(* Logix 5000 project; controller WP_Ottawa_Data_Concentrator_1 vendor 1 type 14 code 167 rev 32.14; software revision 32.04; part 2 of 5 *)
(* tags used below, declared in another part *)
   Break1_Length : DINT;
   Break2_Length : DINT;
   Lunch_Length : DINT;
   PreviousCount : DINT;
   Shift_Reset : BOOL;
   Shift_Reset_ONS : BOOL;
   LN31_Current_Shift_Duration_Mins : DINT;
   LN31_Current_Shift_Duration_wBreaks_Mins : DINT;
   LN31_DC_Controlled_Theoretical_Units : BOOL;
   LN31_Schedule : UDT_Current_Status;
   LN31_Schedule_Cycle_Timer : TIMER;
   LN31_Schedule_Max_Break_Duration : DINT;
   LN31_Schedule_Max_Break_Timer : TIMER;
   LN31_Schedule_TAKT : REAL;
   LN31_ScheduleUnits_Produced_from_line : DINT;
   LN31_Theoretical_Units_Counter : COUNTER;
   LN31_Theoretical_Units_Counter_ONS : BOOL;
   LN31_Weekly_Schedule : UDT_Weekly_Schedule;
   LN31_WorkstationsOA : DINT[120];
   null : STRING;
   Previous_Shift_Count : DINT;
(* LN31, continued *)

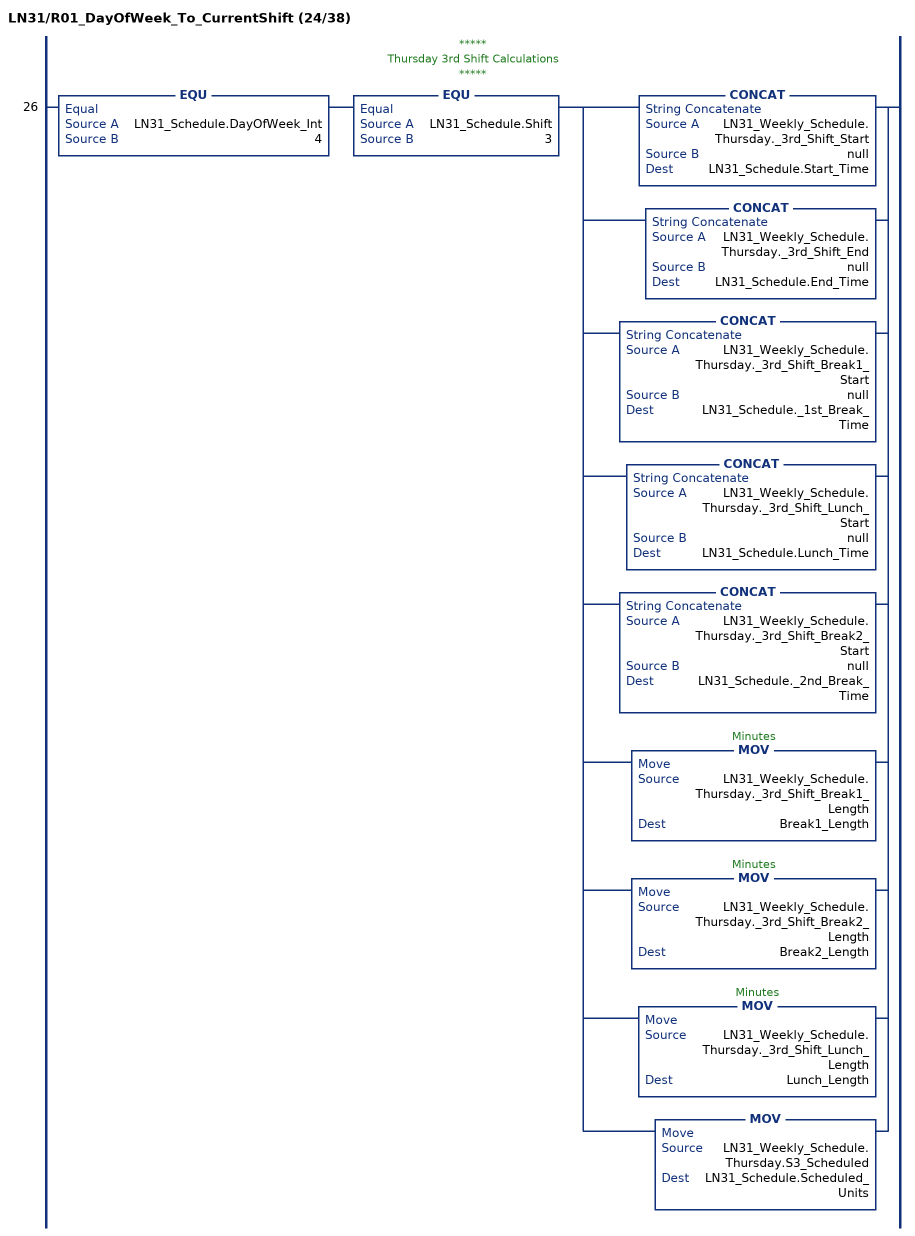
   [picture p24: LN31/R01_DayOfWeek_To_CurrentShift rungs 26-26]
   // *****
   // Thursday 3rd Shift Calculations
   // *****
   26: EQU(LN31_Schedule.DayOfWeek_Int,4)EQU(LN31_Schedule.Shift,3)[CONCAT(LN31_Weekly_Schedule.Thursday._3rd_Shift_Start,null,LN31_Schedule.Start_Time) ,CONCAT(LN31_Weekly_Schedule.Thursday._3rd_Shift_End,null,LN31_Schedule.End_Time) ,CONCAT(LN31_Weekly_Schedule.Thursday._3rd_Shift_Break1_Start,null,LN31_Schedule._1st_Break_Time) ,CONCAT(LN31_Weekly_Schedule.Thursday._3rd_Shift_Lunch_Start,null,LN31_Schedule.Lunch_Time) ,CONCAT(LN31_Weekly_Schedule.Thursday._3rd_Shift_Break2_Start,null,LN31_Schedule._2nd_Break_Time) ,MOV(LN31_Weekly_Schedule.Thursday._3rd_Shift_Break1_Length,Break1_Length) ,MOV(LN31_Weekly_Schedule.Thursday._3rd_Shift_Break2_Length,Break2_Length) ,MOV(LN31_Weekly_Schedule.Thursday._3rd_Shift_Lunch_Length,Lunch_Length) ,MOV(LN31_Weekly_Schedule.Thursday.S3_Scheduled,LN31_Schedule.Scheduled_Units) ];
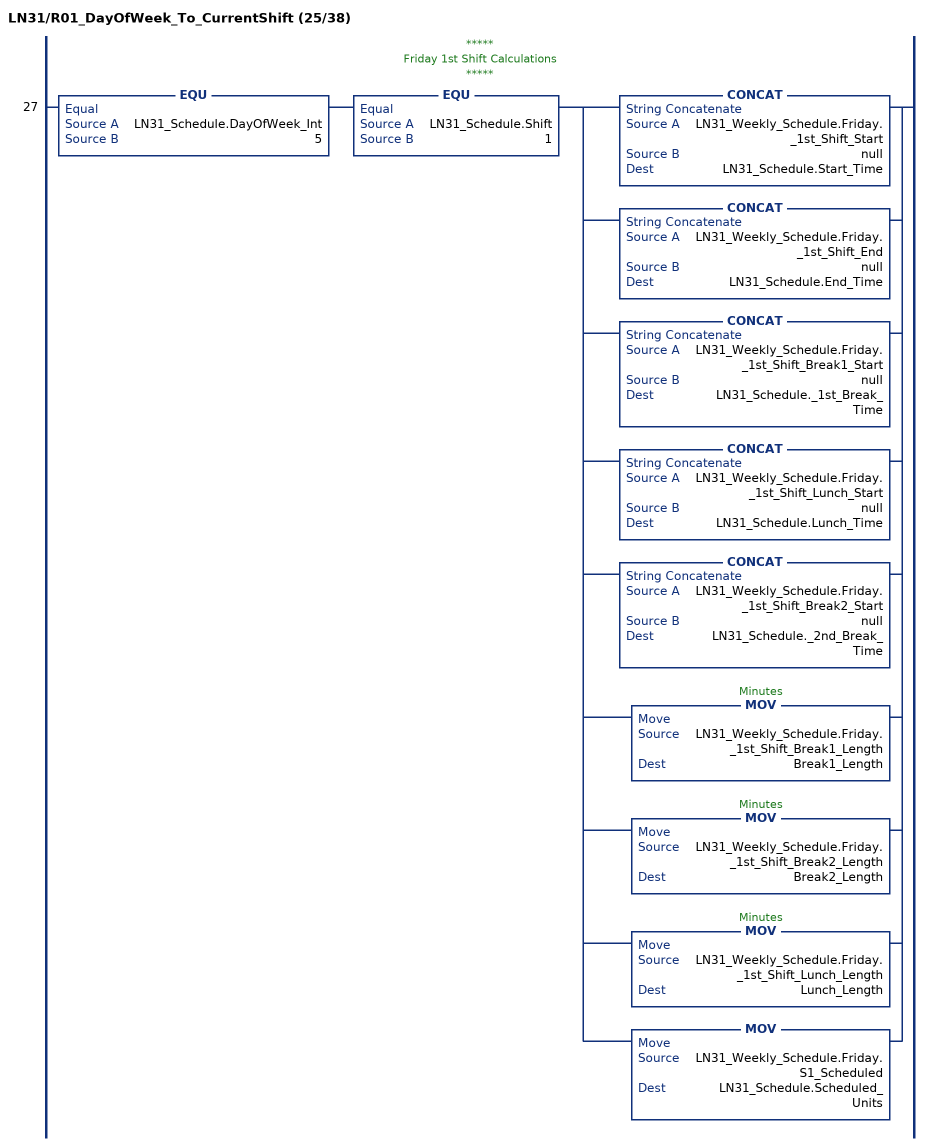
   // *****
   // Friday 1st Shift Calculations
   // *****
   27: EQU(LN31_Schedule.DayOfWeek_Int,5)EQU(LN31_Schedule.Shift,1)[CONCAT(LN31_Weekly_Schedule.Friday._1st_Shift_Start,null,LN31_Schedule.Start_Time) ,CONCAT(LN31_Weekly_Schedule.Friday._1st_Shift_End,null,LN31_Schedule.End_Time) ,CONCAT(LN31_Weekly_Schedule.Friday._1st_Shift_Break1_Start,null,LN31_Schedule._1st_Break_Time) ,CONCAT(LN31_Weekly_Schedule.Friday._1st_Shift_Lunch_Start,null,LN31_Schedule.Lunch_Time) ,CONCAT(LN31_Weekly_Schedule.Friday._1st_Shift_Break2_Start,null,LN31_Schedule._2nd_Break_Time) ,MOV(LN31_Weekly_Schedule.Friday._1st_Shift_Break1_Length,Break1_Length) ,MOV(LN31_Weekly_Schedule.Friday._1st_Shift_Break2_Length,Break2_Length) ,MOV(LN31_Weekly_Schedule.Friday._1st_Shift_Lunch_Length,Lunch_Length) ,MOV(LN31_Weekly_Schedule.Friday.S1_Scheduled,LN31_Schedule.Scheduled_Units) ];
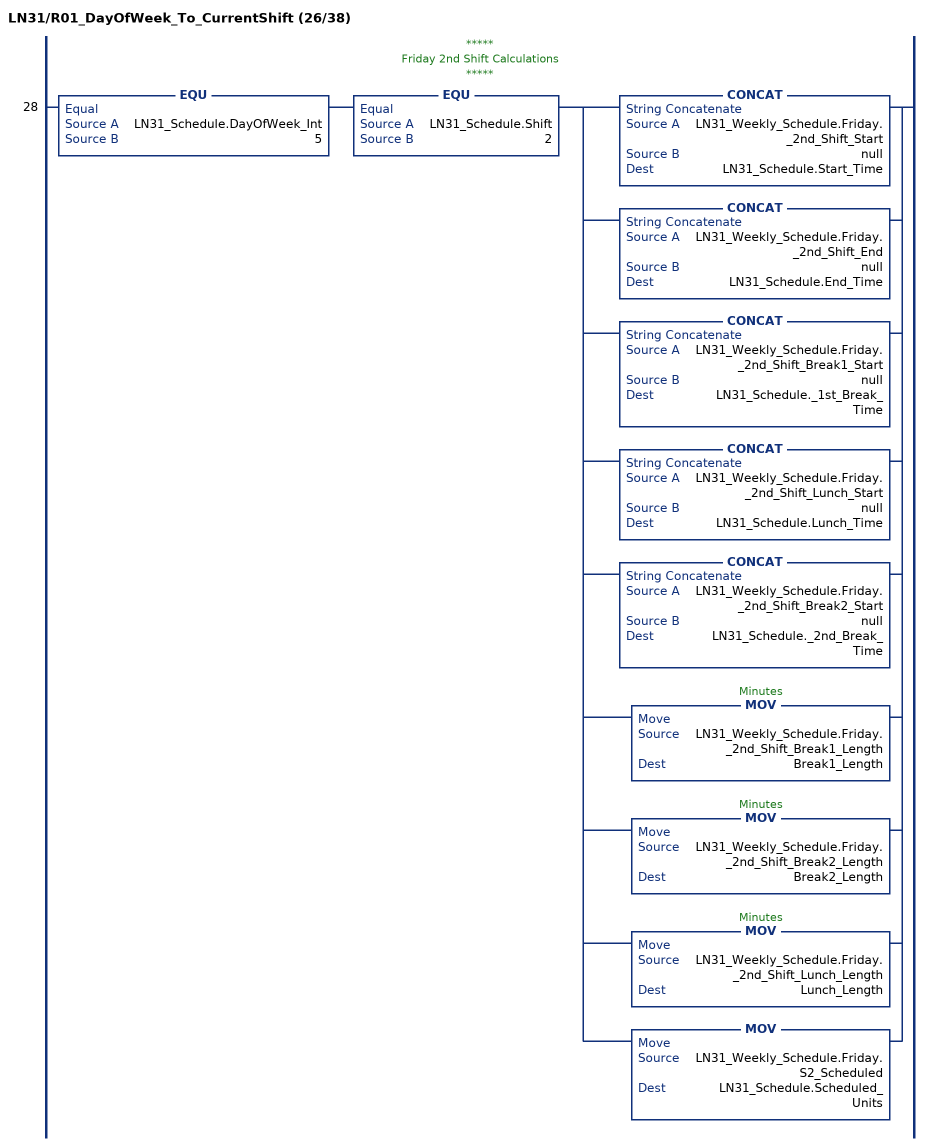
   // *****
   // Friday 2nd Shift Calculations
   // *****
   28: EQU(LN31_Schedule.DayOfWeek_Int,5)EQU(LN31_Schedule.Shift,2)[CONCAT(LN31_Weekly_Schedule.Friday._2nd_Shift_Start,null,LN31_Schedule.Start_Time) ,CONCAT(LN31_Weekly_Schedule.Friday._2nd_Shift_End,null,LN31_Schedule.End_Time) ,CONCAT(LN31_Weekly_Schedule.Friday._2nd_Shift_Break1_Start,null,LN31_Schedule._1st_Break_Time) ,CONCAT(LN31_Weekly_Schedule.Friday._2nd_Shift_Lunch_Start,null,LN31_Schedule.Lunch_Time) ,CONCAT(LN31_Weekly_Schedule.Friday._2nd_Shift_Break2_Start,null,LN31_Schedule._2nd_Break_Time) ,MOV(LN31_Weekly_Schedule.Friday._2nd_Shift_Break1_Length,Break1_Length) ,MOV(LN31_Weekly_Schedule.Friday._2nd_Shift_Break2_Length,Break2_Length) ,MOV(LN31_Weekly_Schedule.Friday._2nd_Shift_Lunch_Length,Lunch_Length) ,MOV(LN31_Weekly_Schedule.Friday.S2_Scheduled,LN31_Schedule.Scheduled_Units) ];
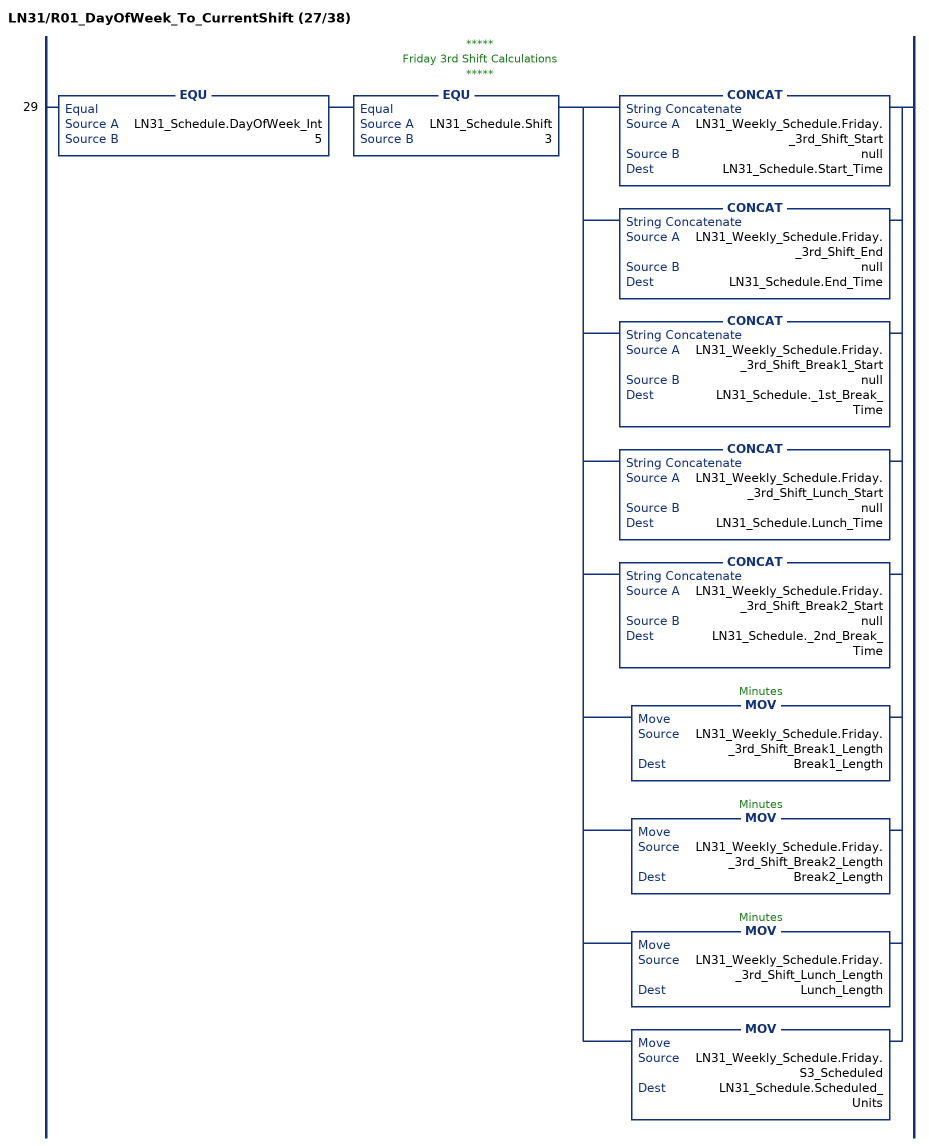
   // *****
   // Friday 3rd Shift Calculations
   // *****
   29: EQU(LN31_Schedule.DayOfWeek_Int,5)EQU(LN31_Schedule.Shift,3)[CONCAT(LN31_Weekly_Schedule.Friday._3rd_Shift_Start,null,LN31_Schedule.Start_Time) ,CONCAT(LN31_Weekly_Schedule.Friday._3rd_Shift_End,null,LN31_Schedule.End_Time) ,CONCAT(LN31_Weekly_Schedule.Friday._3rd_Shift_Break1_Start,null,LN31_Schedule._1st_Break_Time) ,CONCAT(LN31_Weekly_Schedule.Friday._3rd_Shift_Lunch_Start,null,LN31_Schedule.Lunch_Time) ,CONCAT(LN31_Weekly_Schedule.Friday._3rd_Shift_Break2_Start,null,LN31_Schedule._2nd_Break_Time) ,MOV(LN31_Weekly_Schedule.Friday._3rd_Shift_Break1_Length,Break1_Length) ,MOV(LN31_Weekly_Schedule.Friday._3rd_Shift_Break2_Length,Break2_Length) ,MOV(LN31_Weekly_Schedule.Friday._3rd_Shift_Lunch_Length,Lunch_Length) ,MOV(LN31_Weekly_Schedule.Friday.S3_Scheduled,LN31_Schedule.Scheduled_Units) ];
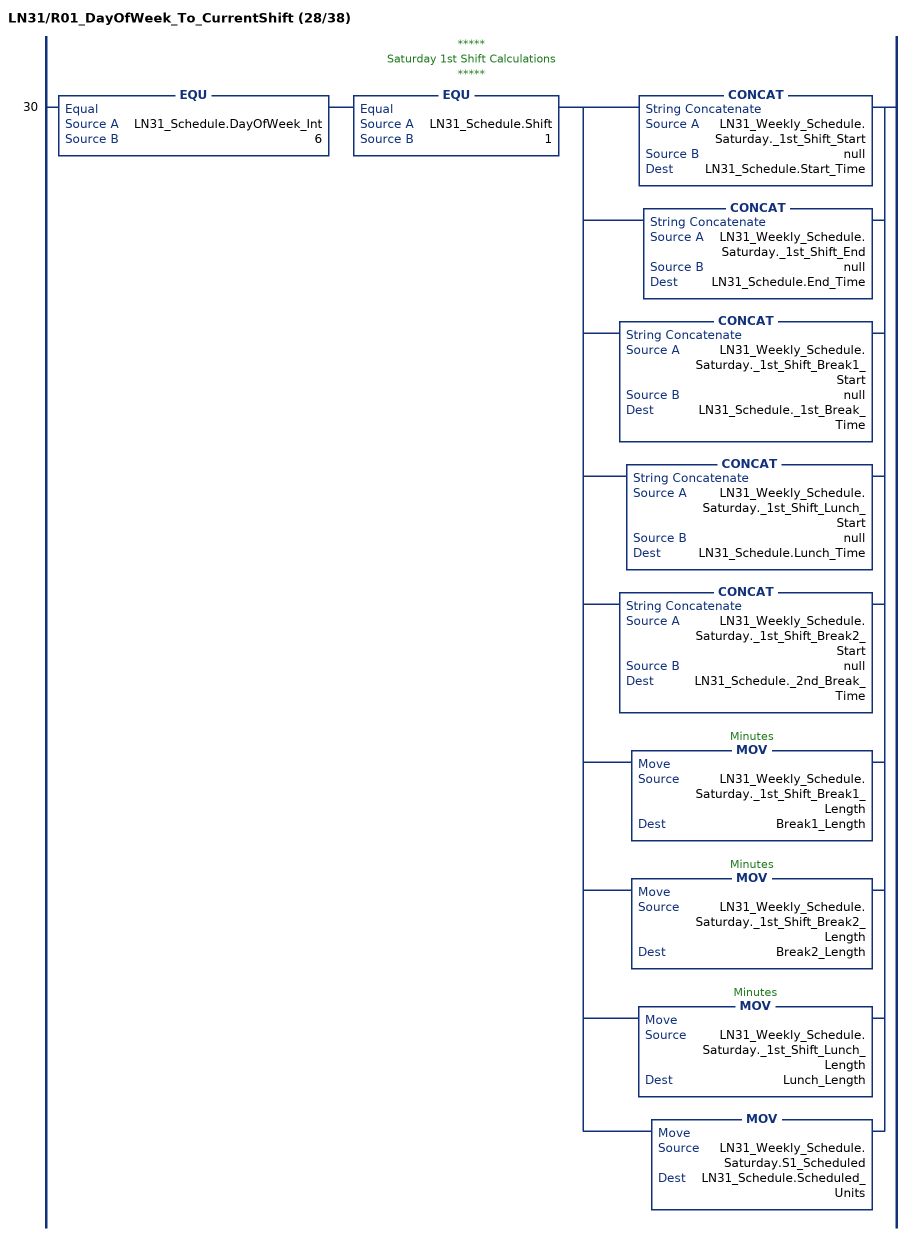
   // *****
   // Saturday 1st Shift Calculations
   // *****
   30: EQU(LN31_Schedule.DayOfWeek_Int,6)EQU(LN31_Schedule.Shift,1)[CONCAT(LN31_Weekly_Schedule.Saturday._1st_Shift_Start,null,LN31_Schedule.Start_Time) ,CONCAT(LN31_Weekly_Schedule.Saturday._1st_Shift_End,null,LN31_Schedule.End_Time) ,CONCAT(LN31_Weekly_Schedule.Saturday._1st_Shift_Break1_Start,null,LN31_Schedule._1st_Break_Time) ,CONCAT(LN31_Weekly_Schedule.Saturday._1st_Shift_Lunch_Start,null,LN31_Schedule.Lunch_Time) ,CONCAT(LN31_Weekly_Schedule.Saturday._1st_Shift_Break2_Start,null,LN31_Schedule._2nd_Break_Time) ,MOV(LN31_Weekly_Schedule.Saturday._1st_Shift_Break1_Length,Break1_Length) ,MOV(LN31_Weekly_Schedule.Saturday._1st_Shift_Break2_Length,Break2_Length) ,MOV(LN31_Weekly_Schedule.Saturday._1st_Shift_Lunch_Length,Lunch_Length) ,MOV(LN31_Weekly_Schedule.Saturday.S1_Scheduled,LN31_Schedule.Scheduled_Units) ];
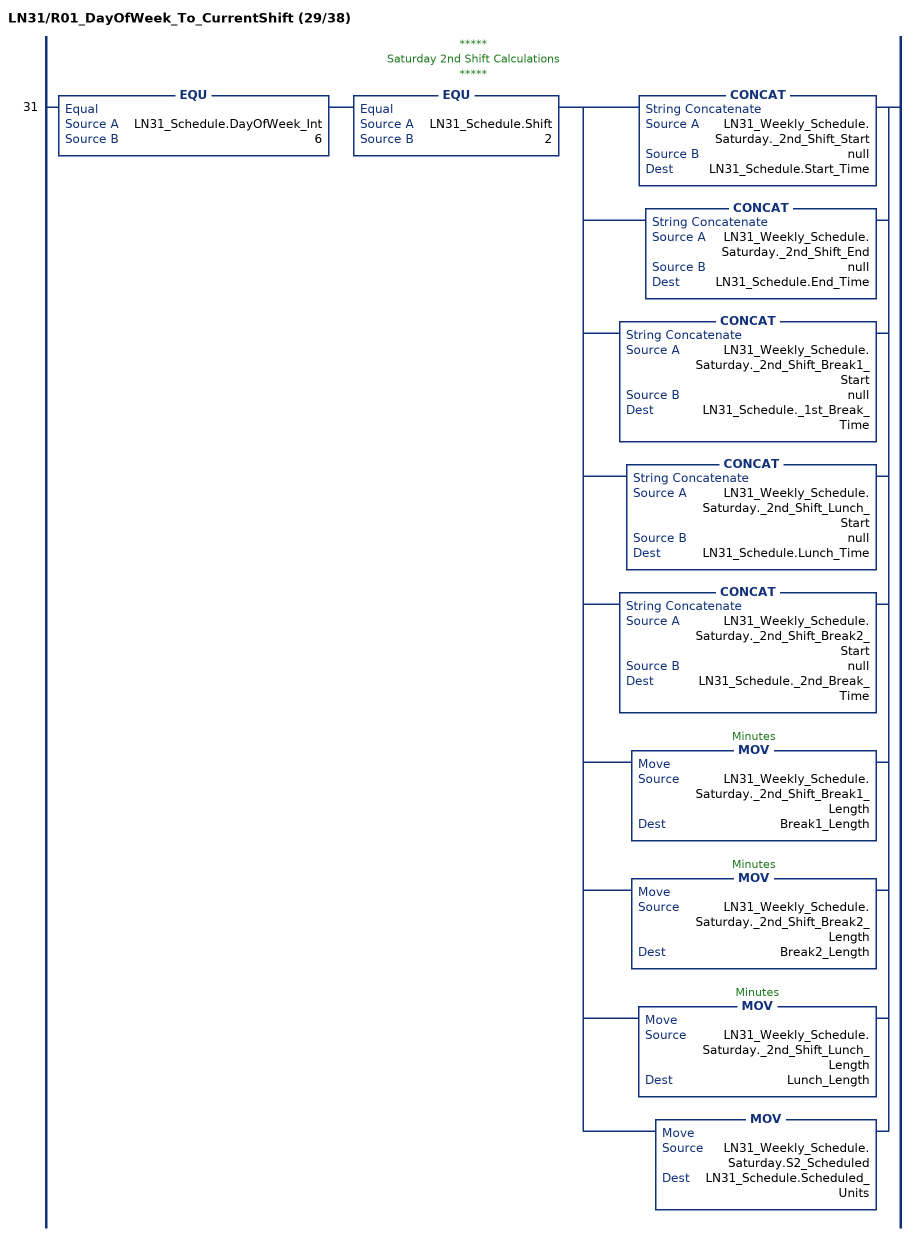
   // *****
   // Saturday 2nd Shift Calculations
   // *****
   31: EQU(LN31_Schedule.DayOfWeek_Int,6)EQU(LN31_Schedule.Shift,2)[CONCAT(LN31_Weekly_Schedule.Saturday._2nd_Shift_Start,null,LN31_Schedule.Start_Time) ,CONCAT(LN31_Weekly_Schedule.Saturday._2nd_Shift_End,null,LN31_Schedule.End_Time) ,CONCAT(LN31_Weekly_Schedule.Saturday._2nd_Shift_Break1_Start,null,LN31_Schedule._1st_Break_Time) ,CONCAT(LN31_Weekly_Schedule.Saturday._2nd_Shift_Lunch_Start,null,LN31_Schedule.Lunch_Time) ,CONCAT(LN31_Weekly_Schedule.Saturday._2nd_Shift_Break2_Start,null,LN31_Schedule._2nd_Break_Time) ,MOV(LN31_Weekly_Schedule.Saturday._2nd_Shift_Break1_Length,Break1_Length) ,MOV(LN31_Weekly_Schedule.Saturday._2nd_Shift_Break2_Length,Break2_Length) ,MOV(LN31_Weekly_Schedule.Saturday._2nd_Shift_Lunch_Length,Lunch_Length) ,MOV(LN31_Weekly_Schedule.Saturday.S2_Scheduled,LN31_Schedule.Scheduled_Units) ];
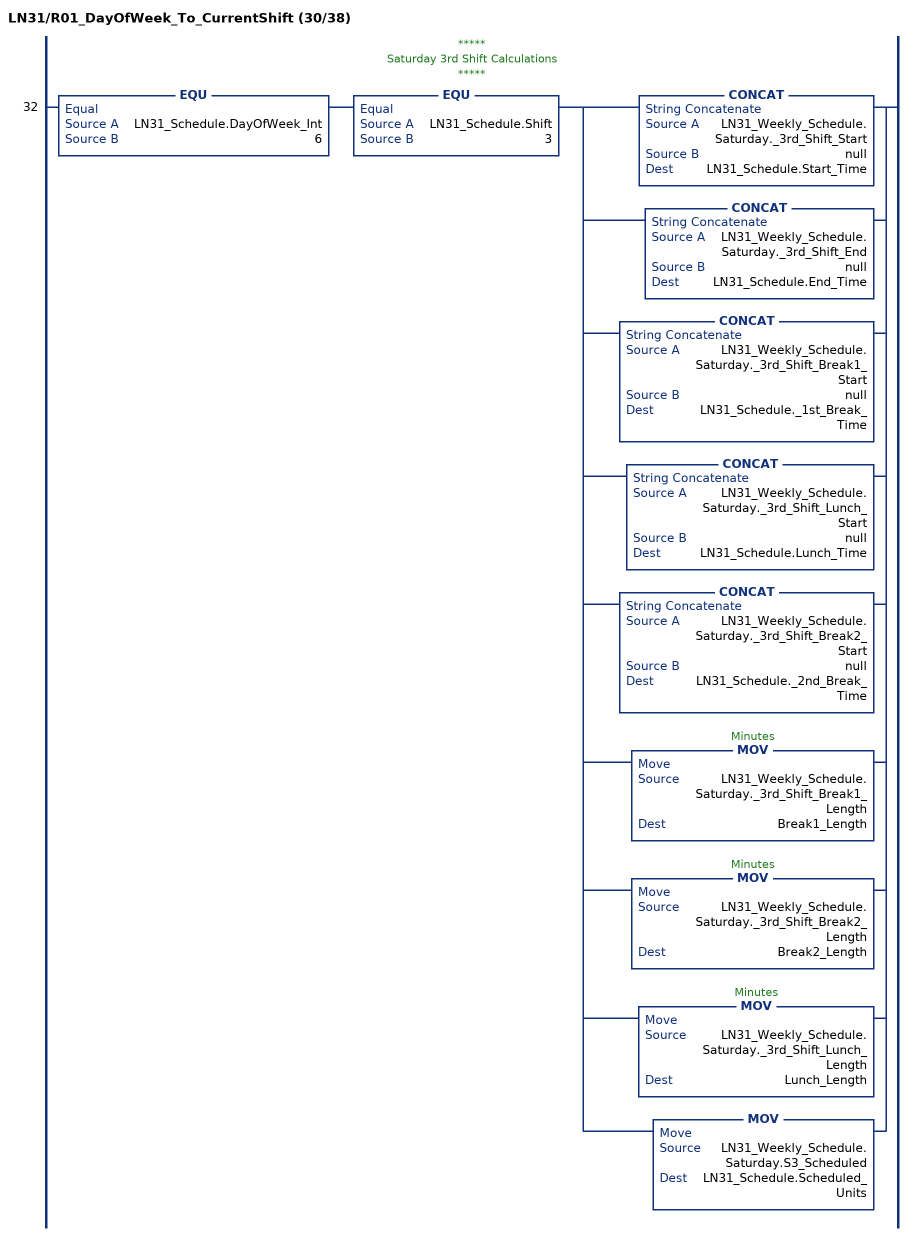
   // *****
   // Saturday 3rd Shift Calculations
   // *****
   32: EQU(LN31_Schedule.DayOfWeek_Int,6)EQU(LN31_Schedule.Shift,3)[CONCAT(LN31_Weekly_Schedule.Saturday._3rd_Shift_Start,null,LN31_Schedule.Start_Time) ,CONCAT(LN31_Weekly_Schedule.Saturday._3rd_Shift_End,null,LN31_Schedule.End_Time) ,CONCAT(LN31_Weekly_Schedule.Saturday._3rd_Shift_Break1_Start,null,LN31_Schedule._1st_Break_Time) ,CONCAT(LN31_Weekly_Schedule.Saturday._3rd_Shift_Lunch_Start,null,LN31_Schedule.Lunch_Time) ,CONCAT(LN31_Weekly_Schedule.Saturday._3rd_Shift_Break2_Start,null,LN31_Schedule._2nd_Break_Time) ,MOV(LN31_Weekly_Schedule.Saturday._3rd_Shift_Break1_Length,Break1_Length) ,MOV(LN31_Weekly_Schedule.Saturday._3rd_Shift_Break2_Length,Break2_Length) ,MOV(LN31_Weekly_Schedule.Saturday._3rd_Shift_Lunch_Length,Lunch_Length) ,MOV(LN31_Weekly_Schedule.Saturday.S3_Scheduled,LN31_Schedule.Scheduled_Units) ];
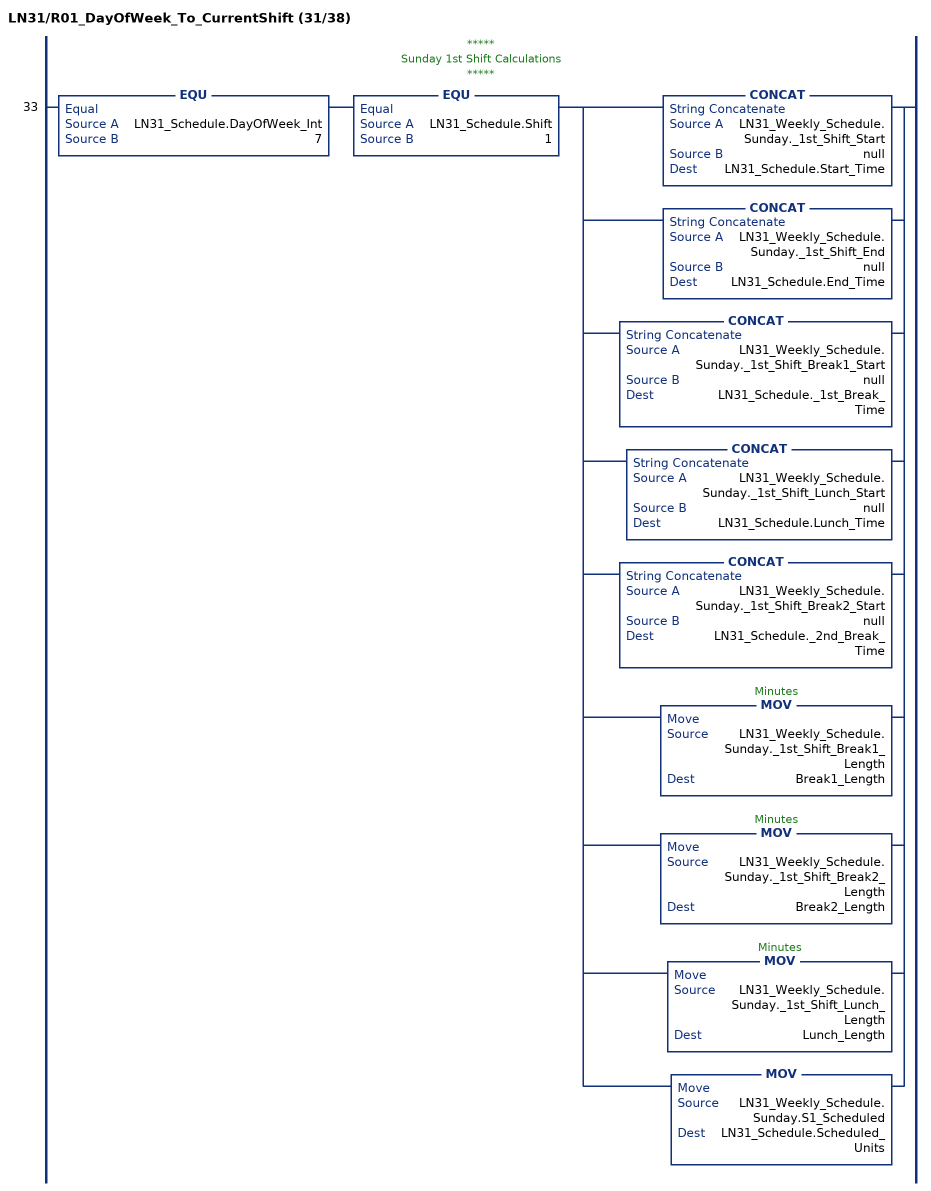
   // *****
   // Sunday 1st Shift Calculations
   // *****
   33: EQU(LN31_Schedule.DayOfWeek_Int,7)EQU(LN31_Schedule.Shift,1)[CONCAT(LN31_Weekly_Schedule.Sunday._1st_Shift_Start,null,LN31_Schedule.Start_Time) ,CONCAT(LN31_Weekly_Schedule.Sunday._1st_Shift_End,null,LN31_Schedule.End_Time) ,CONCAT(LN31_Weekly_Schedule.Sunday._1st_Shift_Break1_Start,null,LN31_Schedule._1st_Break_Time) ,CONCAT(LN31_Weekly_Schedule.Sunday._1st_Shift_Lunch_Start,null,LN31_Schedule.Lunch_Time) ,CONCAT(LN31_Weekly_Schedule.Sunday._1st_Shift_Break2_Start,null,LN31_Schedule._2nd_Break_Time) ,MOV(LN31_Weekly_Schedule.Sunday._1st_Shift_Break1_Length,Break1_Length) ,MOV(LN31_Weekly_Schedule.Sunday._1st_Shift_Break2_Length,Break2_Length) ,MOV(LN31_Weekly_Schedule.Sunday._1st_Shift_Lunch_Length,Lunch_Length) ,MOV(LN31_Weekly_Schedule.Sunday.S1_Scheduled,LN31_Schedule.Scheduled_Units) ];
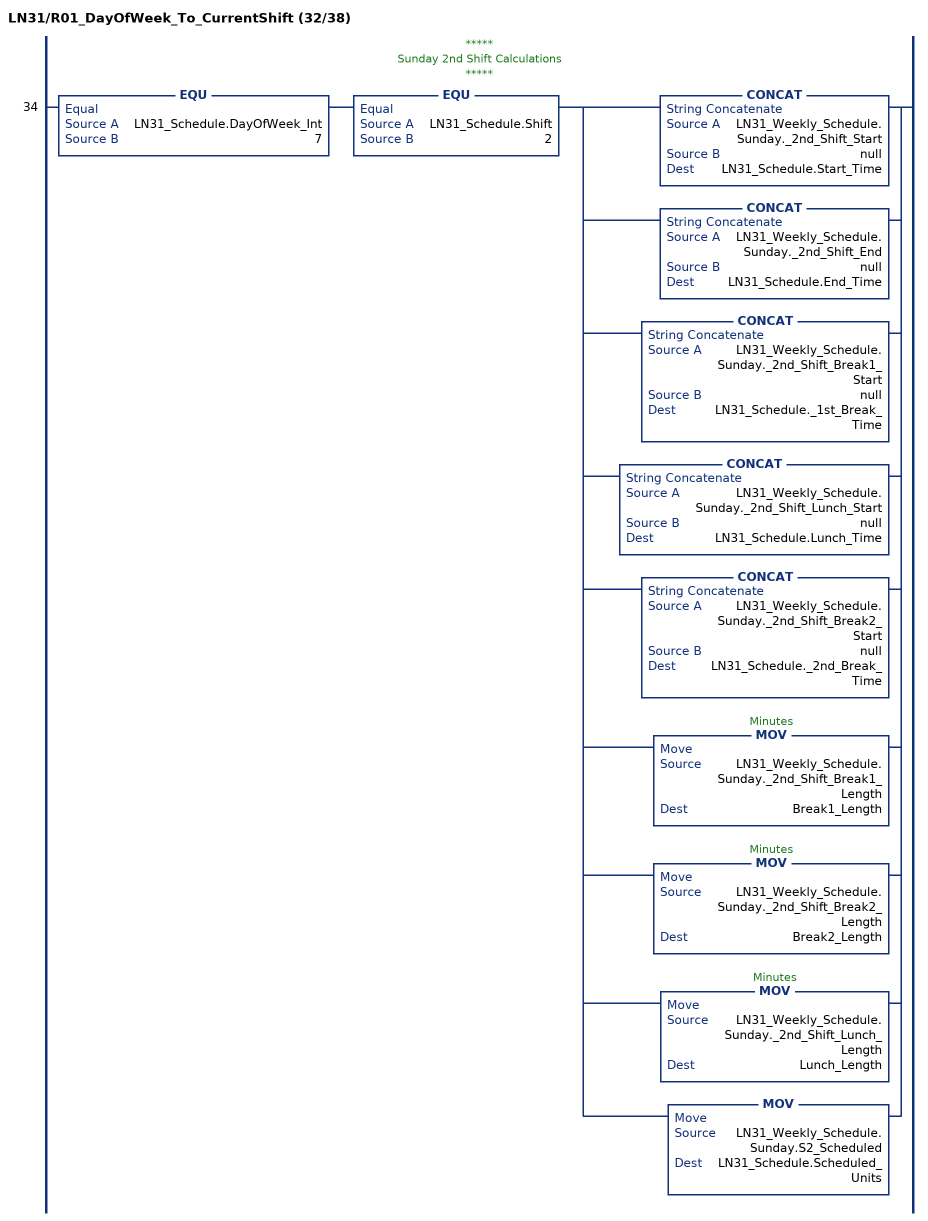
   // *****
   // Sunday 2nd Shift Calculations
   // *****
   34: EQU(LN31_Schedule.DayOfWeek_Int,7)EQU(LN31_Schedule.Shift,2)[CONCAT(LN31_Weekly_Schedule.Sunday._2nd_Shift_Start,null,LN31_Schedule.Start_Time) ,CONCAT(LN31_Weekly_Schedule.Sunday._2nd_Shift_End,null,LN31_Schedule.End_Time) ,CONCAT(LN31_Weekly_Schedule.Sunday._2nd_Shift_Break1_Start,null,LN31_Schedule._1st_Break_Time) ,CONCAT(LN31_Weekly_Schedule.Sunday._2nd_Shift_Lunch_Start,null,LN31_Schedule.Lunch_Time) ,CONCAT(LN31_Weekly_Schedule.Sunday._2nd_Shift_Break2_Start,null,LN31_Schedule._2nd_Break_Time) ,MOV(LN31_Weekly_Schedule.Sunday._2nd_Shift_Break1_Length,Break1_Length) ,MOV(LN31_Weekly_Schedule.Sunday._2nd_Shift_Break2_Length,Break2_Length) ,MOV(LN31_Weekly_Schedule.Sunday._2nd_Shift_Lunch_Length,Lunch_Length) ,MOV(LN31_Weekly_Schedule.Sunday.S2_Scheduled,LN31_Schedule.Scheduled_Units) ];
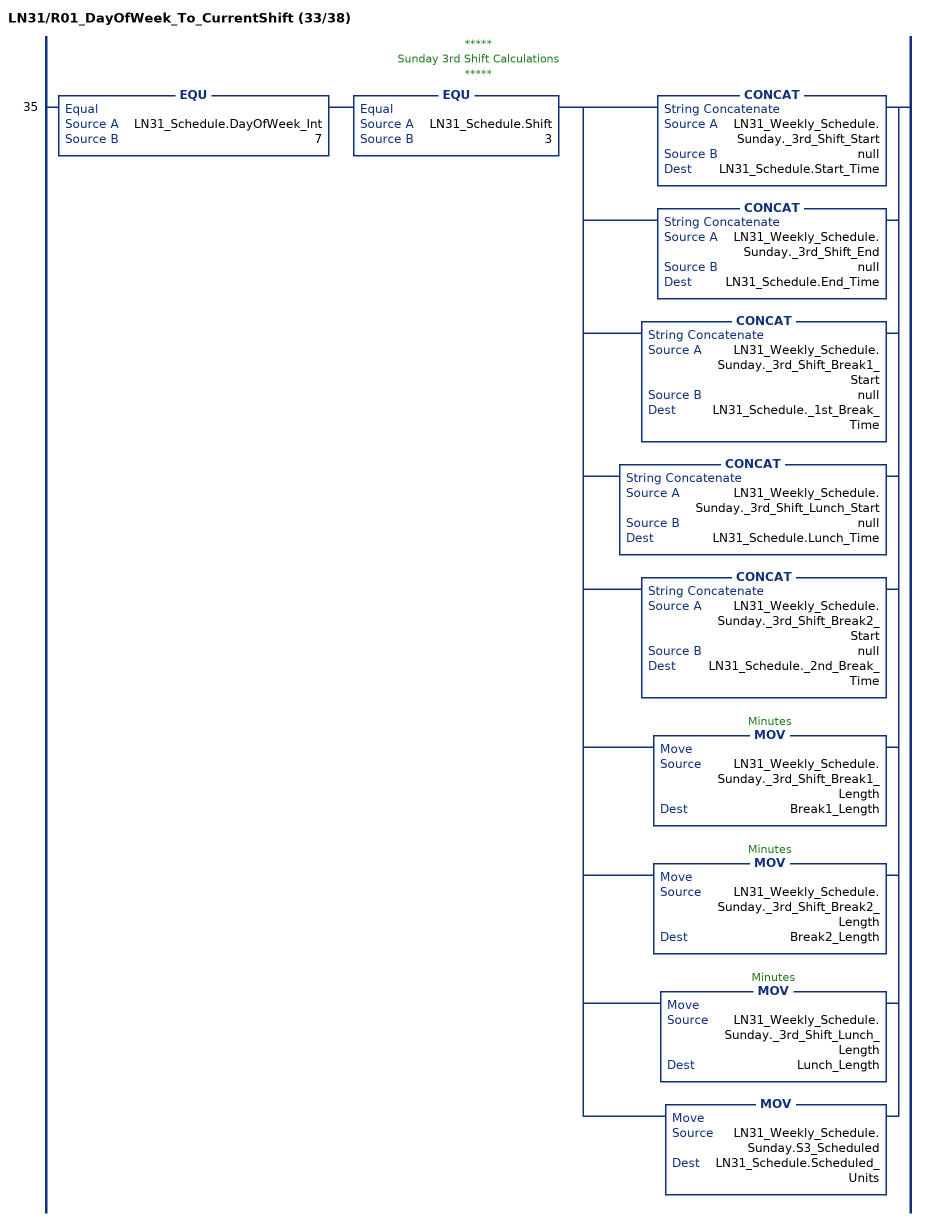
   // *****
   // Sunday 3rd Shift Calculations
   // *****
   35: EQU(LN31_Schedule.DayOfWeek_Int,7)EQU(LN31_Schedule.Shift,3)[CONCAT(LN31_Weekly_Schedule.Sunday._3rd_Shift_Start,null,LN31_Schedule.Start_Time) ,CONCAT(LN31_Weekly_Schedule.Sunday._3rd_Shift_End,null,LN31_Schedule.End_Time) ,CONCAT(LN31_Weekly_Schedule.Sunday._3rd_Shift_Break1_Start,null,LN31_Schedule._1st_Break_Time) ,CONCAT(LN31_Weekly_Schedule.Sunday._3rd_Shift_Lunch_Start,null,LN31_Schedule.Lunch_Time) ,CONCAT(LN31_Weekly_Schedule.Sunday._3rd_Shift_Break2_Start,null,LN31_Schedule._2nd_Break_Time) ,MOV(LN31_Weekly_Schedule.Sunday._3rd_Shift_Break1_Length,Break1_Length) ,MOV(LN31_Weekly_Schedule.Sunday._3rd_Shift_Break2_Length,Break2_Length) ,MOV(LN31_Weekly_Schedule.Sunday._3rd_Shift_Lunch_Length,Lunch_Length) ,MOV(LN31_Weekly_Schedule.Sunday.S3_Scheduled,LN31_Schedule.Scheduled_Units) ];
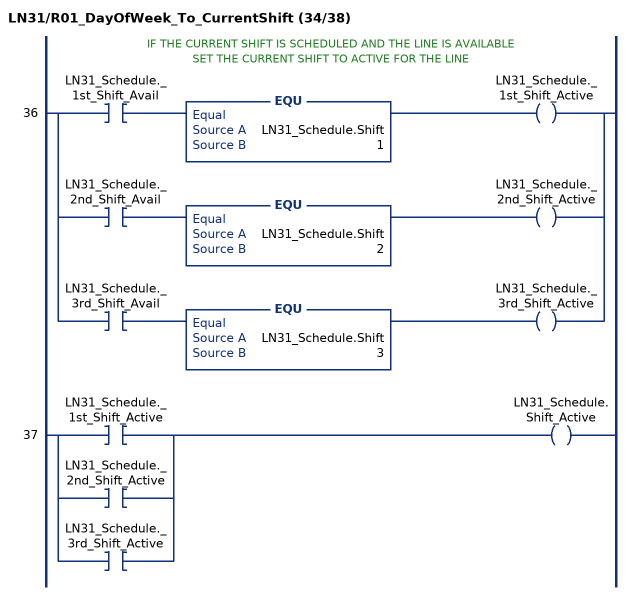
   // IF THE CURRENT SHIFT IS SCHEDULED AND THE LINE IS AVAILABLE
   // SET THE CURRENT SHIFT TO ACTIVE FOR THE LINE
   36: [XIC(LN31_Schedule._1st_Shift_Avail) EQU(LN31_Schedule.Shift,1) OTE(LN31_Schedule._1st_Shift_Active) ,XIC(LN31_Schedule._2nd_Shift_Avail) EQU(LN31_Schedule.Shift,2) OTE(LN31_Schedule._2nd_Shift_Active) ,XIC(LN31_Schedule._3rd_Shift_Avail) EQU(LN31_Schedule.Shift,3) OTE(LN31_Schedule._3rd_Shift_Active) ];
   37: [XIC(LN31_Schedule._1st_Shift_Active) ,XIC(LN31_Schedule._2nd_Shift_Active) ,XIC(LN31_Schedule._3rd_Shift_Active) ]OTE(LN31_Schedule.Shift_Active);
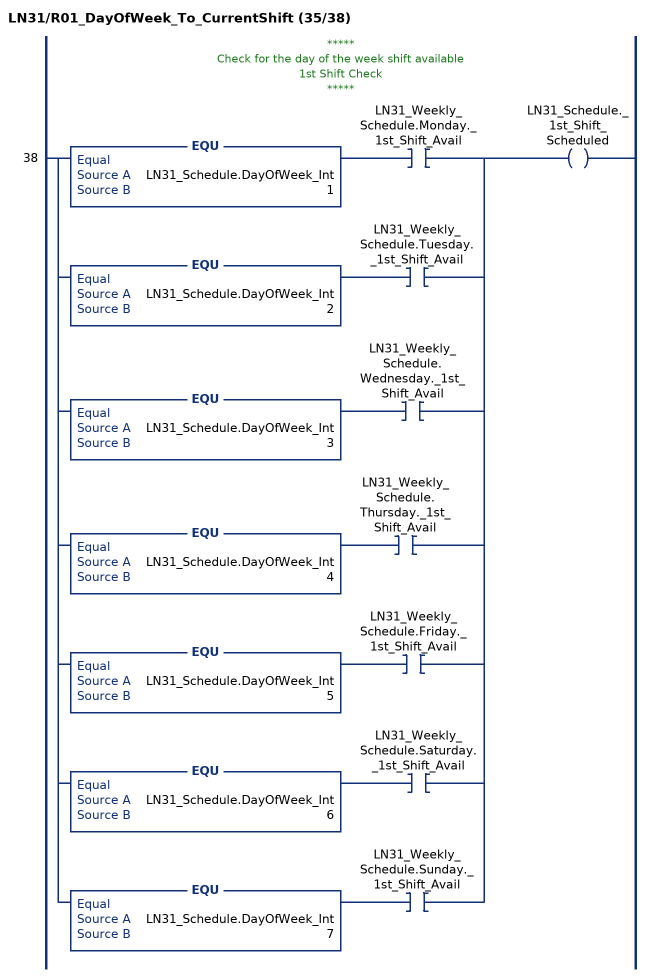
   // *****
   // Check for the day of the week shift available
   // 1st Shift Check
   // *****
   38: [EQU(LN31_Schedule.DayOfWeek_Int,1) XIC(LN31_Weekly_Schedule.Monday._1st_Shift_Avail) ,EQU(LN31_Schedule.DayOfWeek_Int,2) XIC(LN31_Weekly_Schedule.Tuesday._1st_Shift_Avail) ,EQU(LN31_Schedule.DayOfWeek_Int,3) XIC(LN31_Weekly_Schedule.Wednesday._1st_Shift_Avail) ,EQU(LN31_Schedule.DayOfWeek_Int,4) XIC(LN31_Weekly_Schedule.Thursday._1st_Shift_Avail) ,EQU(LN31_Schedule.DayOfWeek_Int,5) XIC(LN31_Weekly_Schedule.Friday._1st_Shift_Avail) ,EQU(LN31_Schedule.DayOfWeek_Int,6) XIC(LN31_Weekly_Schedule.Saturday._1st_Shift_Avail) ,EQU(LN31_Schedule.DayOfWeek_Int,7) XIC(LN31_Weekly_Schedule.Sunday._1st_Shift_Avail) ]OTE(LN31_Schedule._1st_Shift_Scheduled);
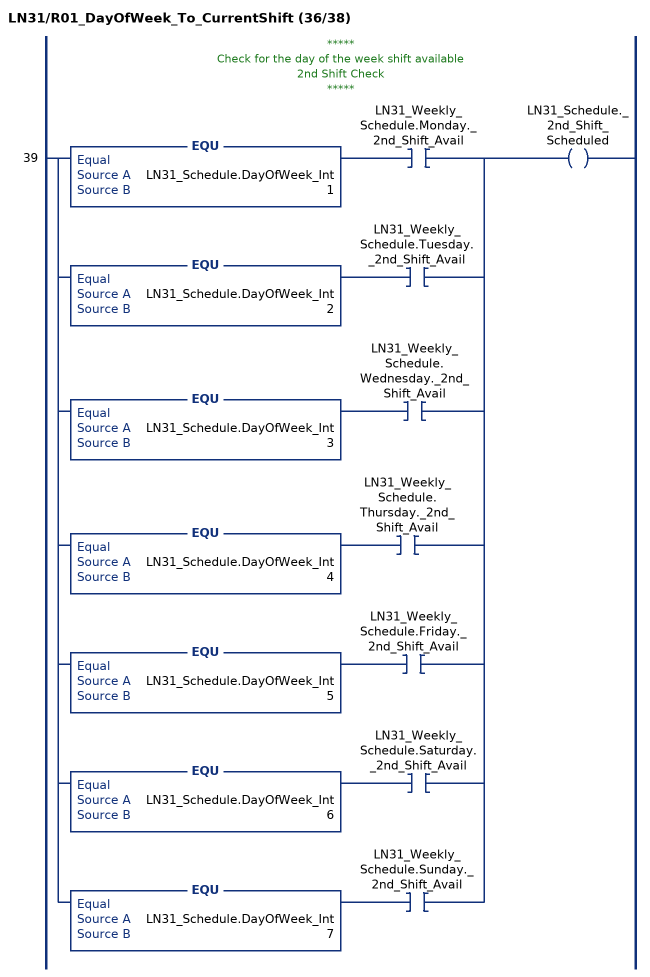
   // *****
   // Check for the day of the week shift available
   // 2nd Shift Check
   // *****
   39: [EQU(LN31_Schedule.DayOfWeek_Int,1) XIC(LN31_Weekly_Schedule.Monday._2nd_Shift_Avail) ,EQU(LN31_Schedule.DayOfWeek_Int,2) XIC(LN31_Weekly_Schedule.Tuesday._2nd_Shift_Avail) ,EQU(LN31_Schedule.DayOfWeek_Int,3) XIC(LN31_Weekly_Schedule.Wednesday._2nd_Shift_Avail) ,EQU(LN31_Schedule.DayOfWeek_Int,4) XIC(LN31_Weekly_Schedule.Thursday._2nd_Shift_Avail) ,EQU(LN31_Schedule.DayOfWeek_Int,5) XIC(LN31_Weekly_Schedule.Friday._2nd_Shift_Avail) ,EQU(LN31_Schedule.DayOfWeek_Int,6) XIC(LN31_Weekly_Schedule.Saturday._2nd_Shift_Avail) ,EQU(LN31_Schedule.DayOfWeek_Int,7) XIC(LN31_Weekly_Schedule.Sunday._2nd_Shift_Avail) ]OTE(LN31_Schedule._2nd_Shift_Scheduled);
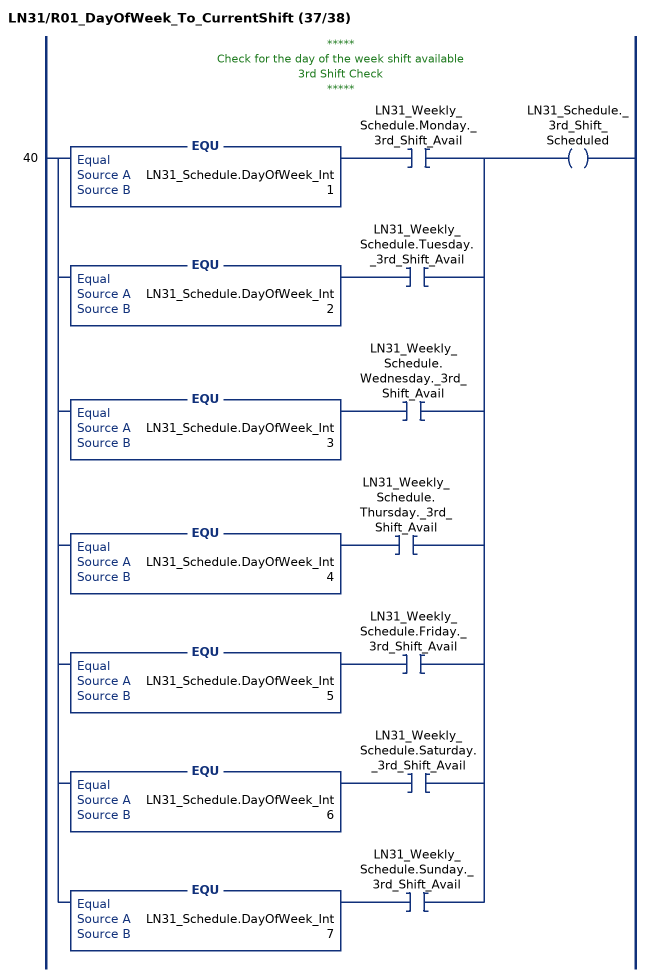
   // *****
   // Check for the day of the week shift available
   // 3rd Shift Check
   // *****
   40: [EQU(LN31_Schedule.DayOfWeek_Int,1) XIC(LN31_Weekly_Schedule.Monday._3rd_Shift_Avail) ,EQU(LN31_Schedule.DayOfWeek_Int,2) XIC(LN31_Weekly_Schedule.Tuesday._3rd_Shift_Avail) ,EQU(LN31_Schedule.DayOfWeek_Int,3) XIC(LN31_Weekly_Schedule.Wednesday._3rd_Shift_Avail) ,EQU(LN31_Schedule.DayOfWeek_Int,4) XIC(LN31_Weekly_Schedule.Thursday._3rd_Shift_Avail) ,EQU(LN31_Schedule.DayOfWeek_Int,5) XIC(LN31_Weekly_Schedule.Friday._3rd_Shift_Avail) ,EQU(LN31_Schedule.DayOfWeek_Int,6) XIC(LN31_Weekly_Schedule.Saturday._3rd_Shift_Avail) ,EQU(LN31_Schedule.DayOfWeek_Int,7) XIC(LN31_Weekly_Schedule.Sunday._3rd_Shift_Avail) ]OTE(LN31_Schedule._3rd_Shift_Scheduled);
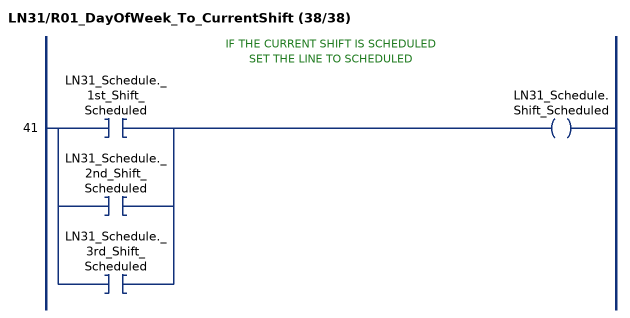
   // IF THE CURRENT SHIFT IS SCHEDULED
   // SET THE LINE TO SCHEDULED
   41: [XIC(LN31_Schedule._1st_Shift_Scheduled) ,XIC(LN31_Schedule._2nd_Shift_Scheduled) ,XIC(LN31_Schedule._3rd_Shift_Scheduled) ]OTE(LN31_Schedule.Shift_Scheduled);
END_ROUTINE

ROUTINE R02_CurrentShift_Calcs   (* ladder *)
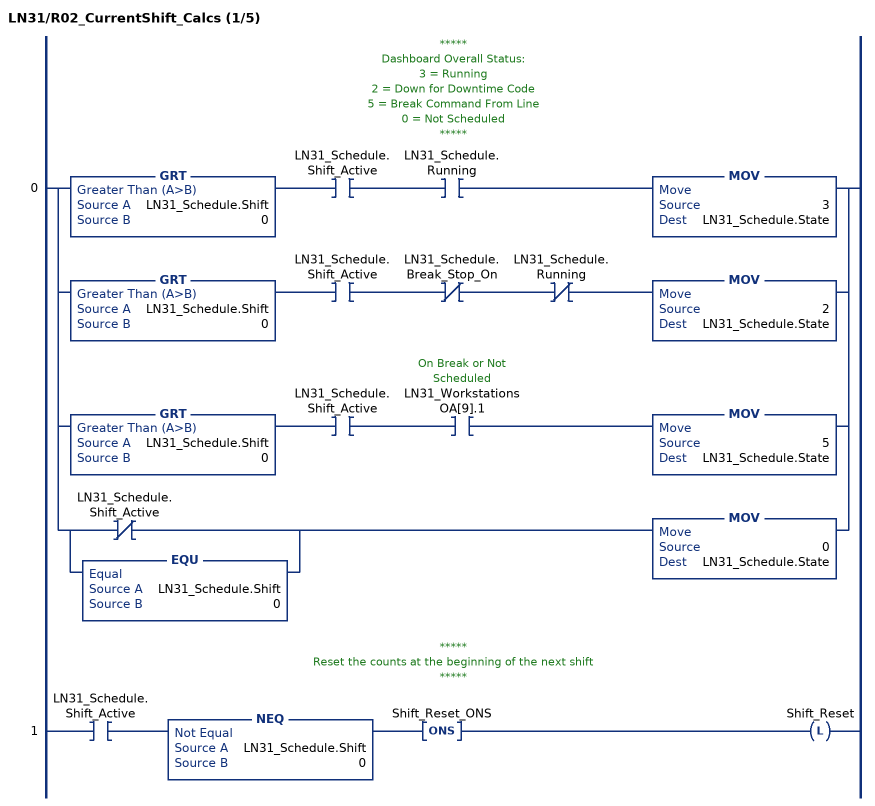
   // *****
   // Dashboard Overall Status:
   // 3 = Running
   // 2 = Down for Downtime Code
   // 5 = Break Command From Line
   // 0 = Not Scheduled
   // *****
   0: [GRT(LN31_Schedule.Shift,0) XIC(LN31_Schedule.Shift_Active) XIC(LN31_Schedule.Running) MOV(3,LN31_Schedule.State) ,GRT(LN31_Schedule.Shift,0) XIC(LN31_Schedule.Shift_Active) XIO(LN31_Schedule.Break_Stop_On) XIO(LN31_Schedule.Running) MOV(2,LN31_Schedule.State) ,GRT(LN31_Schedule.Shift,0) XIC(LN31_Schedule.Shift_Active) XIC(LN31_WorkstationsOA[9].1) MOV(5,LN31_Schedule.State) ,[XIO(LN31_Schedule.Shift_Active) ,EQU(LN31_Schedule.Shift,0) ] MOV(0,LN31_Schedule.State) ];
   // *****
   // Reset the counts at the beginning of the next shift
   // *****
   1: XIC(LN31_Schedule.Shift_Active)NEQ(LN31_Schedule.Shift,0)ONS(Shift_Reset_ONS)OTL(Shift_Reset);
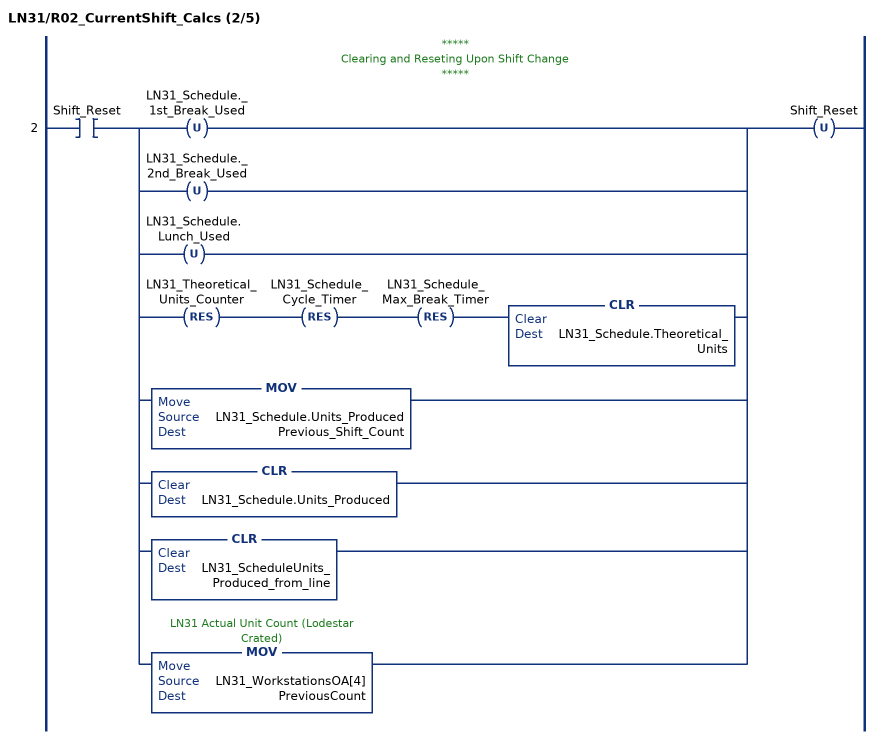
   // *****
   // Clearing and Reseting Upon Shift Change
   // *****
   2: XIC(Shift_Reset)[OTU(LN31_Schedule._1st_Break_Used) ,OTU(LN31_Schedule._2nd_Break_Used) ,OTU(LN31_Schedule.Lunch_Used) ,RES(LN31_Theoretical_Units_Counter) RES(LN31_Schedule_Cycle_Timer) RES(LN31_Schedule_Max_Break_Timer) CLR(LN31_Schedule.Theoretical_Units) ,MOV(LN31_Schedule.Units_Produced,Previous_Shift_Count) ,CLR(LN31_Schedule.Units_Produced) ,CLR(LN31_ScheduleUnits_Produced_from_line) ,MOV(LN31_WorkstationsOA[4],PreviousCount) ]OTU(Shift_Reset);
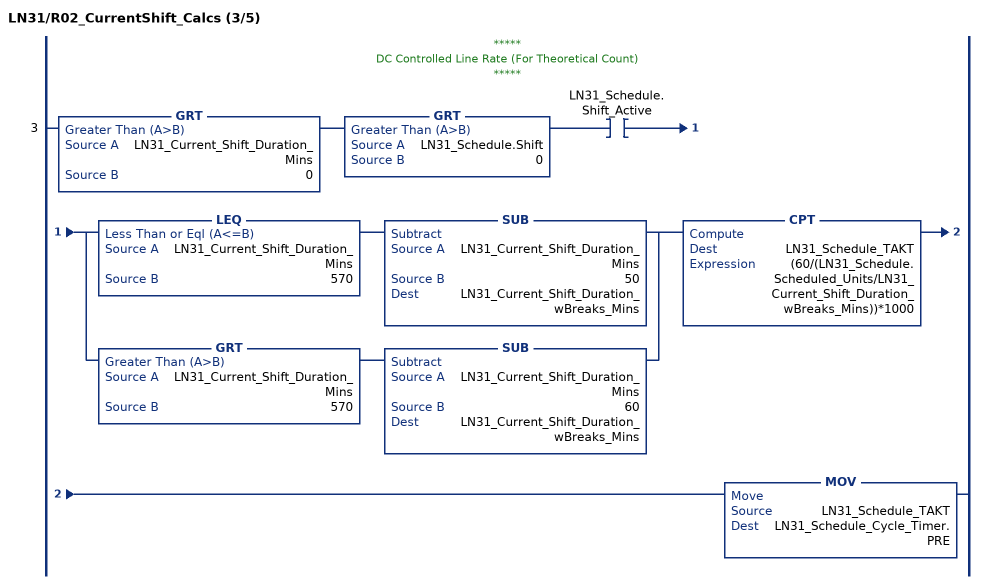
   // *****
   // DC Controlled Line Rate (For Theoretical Count)
   // *****
   3: GRT(LN31_Current_Shift_Duration_Mins,0)GRT(LN31_Schedule.Shift,0)XIC(LN31_Schedule.Shift_Active)[LEQ(LN31_Current_Shift_Duration_Mins,570) SUB(LN31_Current_Shift_Duration_Mins,50,LN31_Current_Shift_Duration_wBreaks_Mins) ,GRT(LN31_Current_Shift_Duration_Mins,570) SUB(LN31_Current_Shift_Duration_Mins,60,LN31_Current_Shift_Duration_wBreaks_Mins) ]CPT(LN31_Schedule_TAKT,(60/(LN31_Schedule.Scheduled_Units/LN31_Current_Shift_Duration_wBreaks_Mins))*1000)MOV(LN31_Schedule_TAKT,LN31_Schedule_Cycle_Timer.PRE);
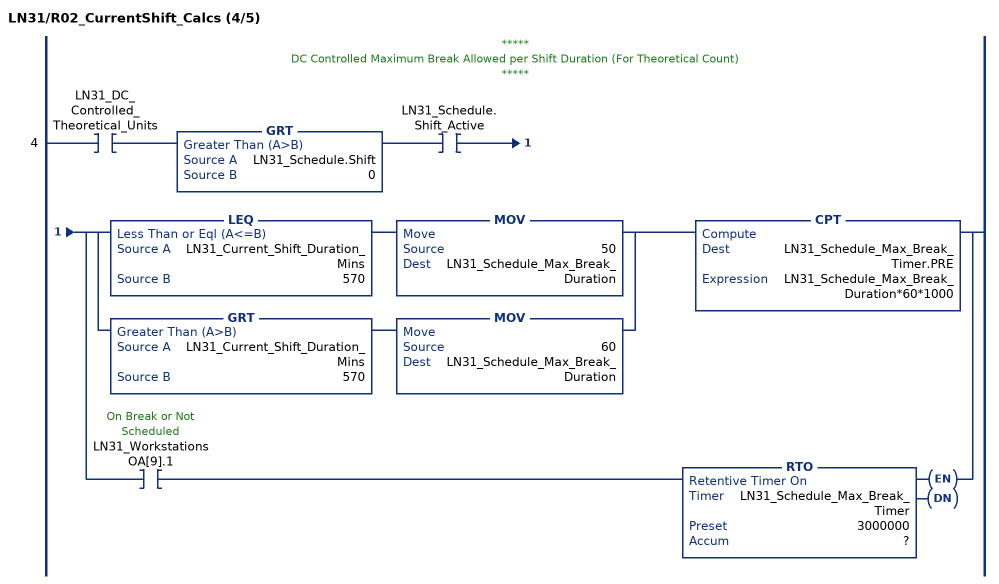
   // *****
   // DC Controlled Maximum Break Allowed per Shift Duration (For Theoretical Count)
   // *****
   4: XIC(LN31_DC_Controlled_Theoretical_Units)GRT(LN31_Schedule.Shift,0)XIC(LN31_Schedule.Shift_Active)[[LEQ(LN31_Current_Shift_Duration_Mins,570) MOV(50,LN31_Schedule_Max_Break_Duration) ,GRT(LN31_Current_Shift_Duration_Mins,570) MOV(60,LN31_Schedule_Max_Break_Duration) ] CPT(LN31_Schedule_Max_Break_Timer.PRE,LN31_Schedule_Max_Break_Duration*60*1000) ,XIC(LN31_WorkstationsOA[9].1) RTO(LN31_Schedule_Max_Break_Timer,?,?) ];
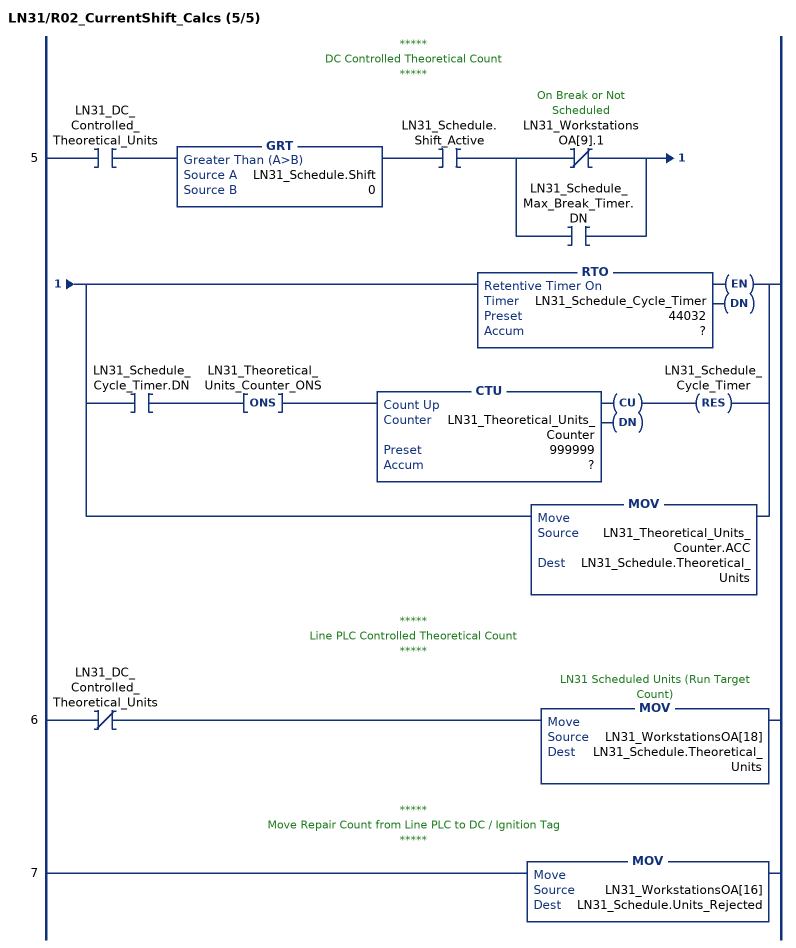
   // *****
   // DC Controlled Theoretical Count
   // *****
   5: XIC(LN31_DC_Controlled_Theoretical_Units)GRT(LN31_Schedule.Shift,0)XIC(LN31_Schedule.Shift_Active)[XIO(LN31_WorkstationsOA[9].1) ,XIC(LN31_Schedule_Max_Break_Timer.DN) ][RTO(LN31_Schedule_Cycle_Timer,?,?) ,XIC(LN31_Schedule_Cycle_Timer.DN) ONS(LN31_Theoretical_Units_Counter_ONS) CTU(LN31_Theoretical_Units_Counter,?,?) RES(LN31_Schedule_Cycle_Timer) ,MOV(LN31_Theoretical_Units_Counter.ACC,LN31_Schedule.Theoretical_Units) ];
   // *****
   // Line PLC Controlled Theoretical Count
   // *****
   6: XIO(LN31_DC_Controlled_Theoretical_Units)MOV(LN31_WorkstationsOA[18],LN31_Schedule.Theoretical_Units);
   // *****
   // Move Repair Count from Line PLC to DC / Ignition Tag
   // *****
   7: MOV(LN31_WorkstationsOA[16],LN31_Schedule.Units_Rejected);
END_ROUTINE
